// TIA Portal V19 export
TYPE "LUC_typeSignalStackByBool"
TITLE = LUC_typeSignalStackPeriphery
// Signal stack type used for a default machine signal stack, includes.
// stored: Access Published
   STRUCT
      red { ExternalWritable := 'False'} : Bool;   // Signal light active- Red
      yellow { ExternalWritable := 'False'} : Bool;   // Signal light active- Yellow
      blue { ExternalWritable := 'False'} : Bool;   // Signal light active- Blue
      green { ExternalWritable := 'False'} : Bool;   // Signal light active - Green
      horn { ExternalWritable := 'False'} : Bool;   // Signal horn - The horn will sound with the configured horn pulse time
      white { ExternalWritable := 'False'} : Bool;   // Signal light active- White
      user1 { ExternalWritable := 'False'} : Bool;   // Signal active- Userdefined 1
      user2 { ExternalWritable := 'False'} : Bool;   // Signal active- Userdefined 2
   END_STRUCT;
END_TYPE
